FUNCTION_BLOCK FB_DeviceBase

VAR
	TagName : STRING;
	Description : STRING;
	TagID : INT;
END_VAR

END_FUNCTION_BLOCK

(* stored: Version 1.1.0.1, ProductVersion 3.1.4024.12
   POU FB_DeviceBase: Id {485bf89f-73f9-4b1b-aaa0-ce1339f868c9}, SpecialFunc None *)
